FUNCTION_BLOCK App2_StripperTempandReactorTemp (* Composite Function Block Type *)
  (* Standard: 61499-2 *)
  (* Version 0.0, 2018-11-06, 4DIAC-IDE, 4DIAC-Consortium *)
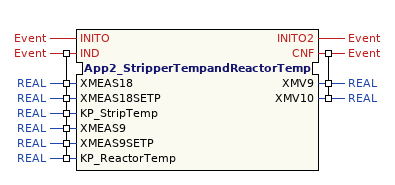
  EVENT_INPUT
    INITO; (* Initialization Request *)
    IND WITH XMEAS18, XMEAS18SETP, XMEAS9, XMEAS9SETP, KP_StripTemp, KP_ReactorTemp; (* Normal Execution Request *)
  END_EVENT
  EVENT_OUTPUT
    INITO2; (* Initialization Confirm *)
    CNF WITH XMV9, XMV10; (* Execution Confirmation *)
  END_EVENT
  VAR_INPUT
    XMEAS18 : REAL;
    XMEAS18SETP : REAL;
    KP_StripTemp : REAL;
    XMEAS9 : REAL;
    XMEAS9SETP : REAL;
    KP_ReactorTemp : REAL;
  END_VAR
  VAR_OUTPUT
    XMV9 : REAL;
    XMV10 : REAL;
  END_VAR
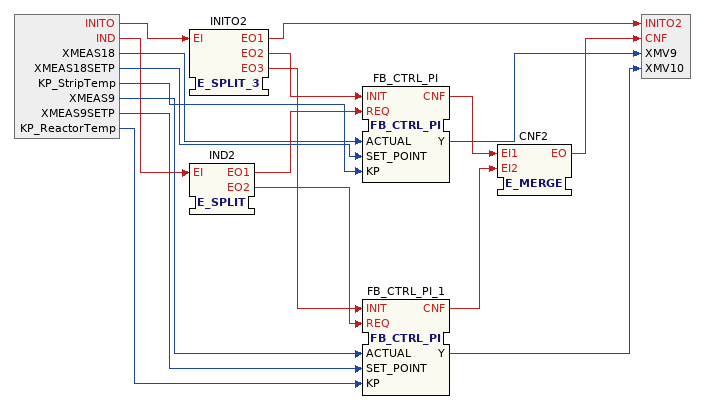
  FBS
    INITO2 : E_SPLIT_3;
    IND2 : E_SPLIT;
    FB_CTRL_PI : FB_CTRL_PI;
    FB_CTRL_PI_1 : FB_CTRL_PI;
    CNF2 : E_MERGE;
  END_FBS
  EVENT_CONNECTIONS
    INITO2.EO1 TO INITO2;
    INITO2.EO2 TO FB_CTRL_PI.INIT;
    INITO2.EO3 TO FB_CTRL_PI_1.INIT;
    IND2.EO1 TO FB_CTRL_PI.REQ;
    IND2.EO2 TO FB_CTRL_PI_1.REQ;
    FB_CTRL_PI.CNF TO CNF2.EI1;
    FB_CTRL_PI_1.CNF TO CNF2.EI2;
    CNF2.EO TO CNF;
    IND TO IND2.EI;
    INITO TO INITO2.EI;
  END_CONNECTIONS
  DATA_CONNECTIONS
    FB_CTRL_PI.Y TO XMV9;
    FB_CTRL_PI_1.Y TO XMV10;
    XMEAS18 TO FB_CTRL_PI.ACTUAL;
    XMEAS18SETP TO FB_CTRL_PI.SET_POINT;
    XMEAS9 TO FB_CTRL_PI_1.ACTUAL;
    XMEAS9SETP TO FB_CTRL_PI_1.SET_POINT;
    KP_StripTemp TO FB_CTRL_PI.KP;
    KP_ReactorTemp TO FB_CTRL_PI_1.KP;
  END_CONNECTIONS
END_FUNCTION_BLOCK
